FUNCTION_BLOCK NextFeedHorizon_HMI (* Service Interface Function Block Type *)
  (* Standard: 61499-2 *)
  (* Version 0.0, 7/15/2026, Schneider Electric, template *)
  PACKAGE SE.Nereda;
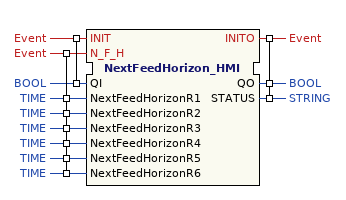
  EVENT_INPUT
    INIT WITH QI;
    N_F_H WITH NextFeedHorizonR1, NextFeedHorizonR2, NextFeedHorizonR3, NextFeedHorizonR4, NextFeedHorizonR5, NextFeedHorizonR6;
  END_EVENT
  EVENT_OUTPUT
    INITO WITH QO, STATUS;
  END_EVENT
  VAR_INPUT
    QI : BOOL;
    NextFeedHorizonR1 : TIME;
    NextFeedHorizonR2 : TIME;
    NextFeedHorizonR3 : TIME;
    NextFeedHorizonR4 : TIME;
    NextFeedHorizonR5 : TIME;
    NextFeedHorizonR6 : TIME;
  END_VAR
  VAR_OUTPUT
    QO : BOOL; (* Event Output Qualifier *)
    STATUS : STRING; (* Service Status *)
  END_VAR
  SERVICE /
    SEQUENCE 
    END_SEQUENCE
  END_SERVICE
END_FUNCTION_BLOCK
